TYPE ST_LIST_CTRL :
STRUCT
  Cmd         : E_LIST_CTRL;
END_STRUCT
END_TYPE

(* stored: Version 1.1.0.1, ProductVersion 3.1.4026.18
   DUT ST_LIST_CTRL: Id {c0b5b920-d3b3-437a-862c-05e0c6120429} *)
